FUNCTION_BLOCK PIOC_Instantaneous_Overcurrent_Logic (* Basic Function Block Type *)
  (* Standard: 61499-2 *)
  (* Version 0.0, 12/10/2023, Cheyan, Schneider Electric, Template *)
  PACKAGE Main;
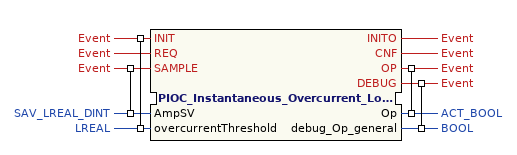
  EVENT_INPUT
    INIT WITH overcurrentThreshold; (* Initialization Request *)
    REQ; (* Normal Execution Request *)
    SAMPLE WITH AmpSV;
  END_EVENT
  EVENT_OUTPUT
    INITO; (* Initialization Confirm *)
    CNF; (* Execution Confirmation *)
    OP WITH Op;
    DEBUG WITH debug_Op_general;
  END_EVENT
  VAR_INPUT
    AmpSV : SAV_LREAL_DINT; (* Input event qualifier *)
    overcurrentThreshold : LREAL;
  END_VAR
  VAR_OUTPUT
    Op : ACT_BOOL;
    debug_Op_general : BOOL;
  END_VAR
  VAR
    overcurrentCounterInternal : DINT := 0;
  END_VAR
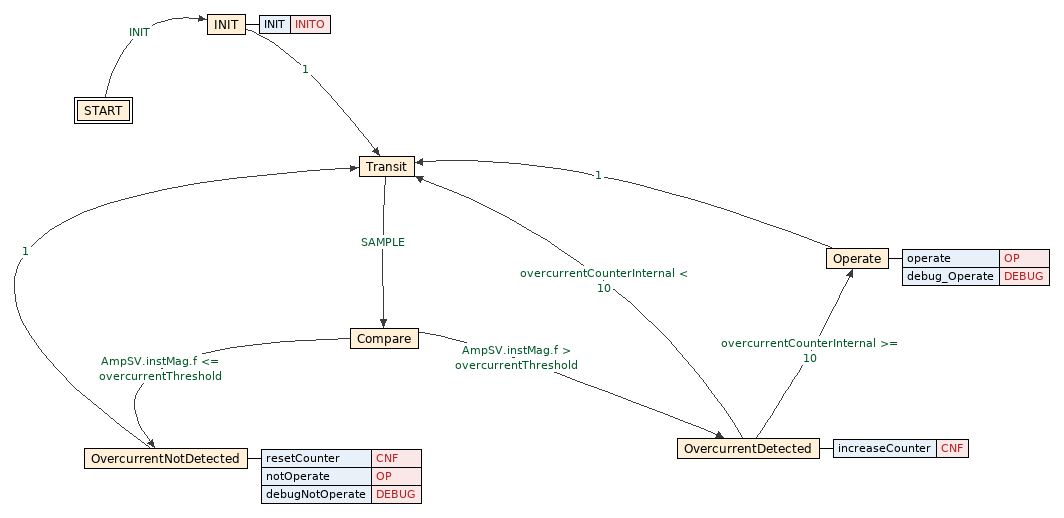
  EC_STATES
    START; (* Initial State *)
    INIT : INIT -> INITO; (* Initialization *)
    Transit; (* Normal execution *)
    OvercurrentNotDetected : resetCounter -> CNF, notOperate -> OP, debugNotOperate -> DEBUG;
    OvercurrentDetected : increaseCounter -> CNF;
    Compare;
    Operate : operate -> OP, debug_Operate -> DEBUG;
  END_STATES
  EC_TRANSITIONS
    START TO INIT := INIT;
    INIT TO Transit := 1;
    Compare TO OvercurrentNotDetected := AmpSV.instMag.f <= overcurrentThreshold;
    Compare TO OvercurrentDetected := AmpSV.instMag.f > overcurrentThreshold;
    Transit TO Compare := SAMPLE;
    OvercurrentNotDetected TO Transit := 1;
    OvercurrentDetected TO Operate := overcurrentCounterInternal >= 10;
    Operate TO Transit := 1;
    OvercurrentDetected TO Transit := overcurrentCounterInternal < 10;
  END_TRANSITIONS
  ALGORITHM INIT IN ST: (* Initialization algorithm *)
;
  END_ALGORITHM
  ALGORITHM resetCounter IN ST: (* Set the overcurrent counter to 0 *)
;

overcurrentCounterInternal := 0;
  END_ALGORITHM
  ALGORITHM increaseCounter IN ST: (* increase the internal overcurrent counter *)
;

overcurrentCounterInternal := overcurrentCounterInternal + 1;
  END_ALGORITHM
  ALGORITHM operate IN ST: (* When an overcurrent fault is detected (after detection of 10 overcurrent measurement), Op_general is set to FALSE *)
;

Op.general := TRUE;
  END_ALGORITHM
  ALGORITHM notOperate IN ST:
;

Op.general := FALSE;
  END_ALGORITHM
  ALGORITHM debug_Operate IN ST:
;

debug_Op_general := TRUE;
  END_ALGORITHM
  ALGORITHM debugNotOperate IN ST:
;

debug_Op_general := FALSE;
  END_ALGORITHM
END_FUNCTION_BLOCK
